(* IEC 61131-3 sources: AutomationLab/ConveyorObject, 5 files *)

(* ---- ConveyorType.st ---- *)
TYPE ConveyorType:
STRUCT
	// Коробка на конце ленты (от оптического датчика)
	BoxOnEndPosition: BOOL := FALSE;
	// Команда на вращение ленты
	ComRotateBelt: BOOL := FALSE;
END_STRUCT
END_TYPE

(* ---- ConveyorMain.st ---- *)
FUNCTION_BLOCK ConveyorMain
VAR
    hardIn: HardwareInput;
    logic: LogicDevice;
    hardOut: HardwareOutput;
    hmi: HMIInterface;
END_VAR

// ============================================
// ЧИСТЫЙ ОРКЕСТРАТОР КОНВЕЙЕРА
// ============================================
// НЕ ИСПОЛЬЗУЕТ GVL. Только соединяет блоки:
// Hardware -> LogicDevice -> HardwareOutput -> HMIInterface
// ============================================

// Шаг 1: Hardware читает датчики из GVL -> BoxOnStart/BoxOnEnd
hardIn();

// Шаг 2: LogicDevice вычисляет команду (RS-триггер с самоподхватом)
logic(BoxOnStart:= hardIn.BoxOnStart,
      BoxOnEnd:= hardIn.BoxOnEnd);

// Шаг 3: HardwareOutput пишет команду на двигатель в GVL
hardOut(ComRotate:= logic.ComRotate);

// Шаг 4: HMIInterface зажигает лампочку на панели
hmi(BeltRun:= logic.ComRotate);

(* ---- HardwareInput.st ---- *)
FUNCTION_BLOCK HardwareInput
VAR_OUTPUT
    // Коробка обнаружена на старте (инвертированный НЗ датчик)
    BoxOnStart: BOOL;
    // Коробка обнаружена в конце (инвертированный НЗ датчик)
    BoxOnEnd: BOOL;
END_VAR

// ============================================
// БЛОК ЧТЕНИЯ АППАРАТУРЫ (ЖЕЛЕЗО — ВХОД)
// ============================================
// Отвечает только за чтение физических датчиков.
// Не пишет в GVL — это делает HardwareOutput.
// ============================================

// Чтение НЗ датчиков (инверсия в активный уровень)
BoxOnStart := NOT GVL.DI_SensorA;
BoxOnEnd   := NOT GVL.DI_SensorB;

(* ---- HardwareOutput.st ---- *)
FUNCTION_BLOCK HardwareOutput
VAR_INPUT
    // Команда на вращение ленты от логического блока
    ComRotate: BOOL;
END_VAR

// ============================================
// БЛОК ЗАПИСИ НА АППАРАТУРУ (ЖЕЛЕЗО — ВЫХОД)
// ============================================
// Отвечает за запись команд управления на физические выходы ПЛК.
// Не читает GVL — это делает Hardware (Input).
// ============================================

// Запись команды на двигатель
GVL.DO_ComMotor := ComRotate;

(* ---- HMIInterface.st ---- *)
FUNCTION_BLOCK HMIInterface
VAR_INPUT
    // Сигнал: лента конвейера работает
    BeltRun: BOOL;
END_VAR

// ============================================
// БЛОК СОПРЯЖЕНИЯ С ИНТЕРФЕЙСОМ ОПЕРАТОРА
// ============================================
// Отвечает за:
// 1. Индикацию состояния конвейера на панели оператора
// 2. В будущем: чтение кнопок оператора
// ============================================

// Лампочка "Лента работает" горит, пока BeltRun = TRUE
GVL.DO_LampWork := BeltRun;
